Universal Robots PolyScope program: verticalMove_external.urp

Program verticalMove_external (installation=default directory=/ursim/programs createdIn=5.19.0 lastSavedIn=5.19.0 robotSerialNumber=20195599999)
Calibrated DH parameters: a=[0, -0.425, -0.3922, 0, 0, 0]; d=[0.1625, 0, 0, 0.1333, 0.0997, 0.0996]; alpha=[1.570796, 0, 0, 1.570796, -1.570796, 0]; deltaTheta=[0, 0, 0, 0, 0, 0]
InitVariablesNode
BeforeStart
  setp := p[0.286,0,0.6,0,1.75,0]
Robot Program (runOnlyOnce=false)
  Script: reset_world_model()
  Script: add_frame("vTCP", p[0.286,0,0.690,0,1.57,0],"world")
  Script: thread move_vTCPThread(): move_vTCP() end
  Script: movej("vTCP")
  Script: frame_tracking_enable("world")
  Script: thrd = run move_vTCPThread()
  Loop Forever
    Script: movel(struct(pose=p[0,0.2,0,0,0,0],frame ="vTCP"), v= 0.1)
    Script: movel(struct(pose=p[0,-0.2,0,0,0,0],frame ="vTCP"), v=0.1)
SubProgram SubProgram_1 (keepSynchronizedWithDisk=false)
  tmp := p[0,0,0,0,0,0]
  tmp := p[0,0,0,0,0,0]
  Loop Forever
    Script: tmp[0] = read_input_float_register(0)
    Script: tmp[1] = read_input_float_register(1)
    Script: tmp[2] = read_input_float_register(2)
    Script: tmp[3] = read_input_float_register(3)
    Script: tmp[4] = read_input_float_register(4)
    Script: tmp[5] = read_input_float_register(5)
    If tmp≠setp
      setp := tmp
      Popup Message (haltProgram=false inputType=Variable) variable=setp
    Script: sync()
SubProgram move_vTCP (keepSynchronizedWithDisk=false)
  Loop Forever
    Script: move_frame("vTCP", p[0.286,0,setp[2],0,1.57,0],"world")
    Script: sync()
